Yaskawa INFORM job: R1_W27-A4(90,180)_KM_OKR2.JBI

/JOB
//NAME R1_W27-A4(90,180)_KM_OKR2
///FOLDERNAME KRIS-SCIANA
//POS
///NPOS 118,118,0,4,0,0
///TOOL 0
///POSTYPE PULSE
///PULSE
C00000=32571,-80067,-84751,-11816,58952,90735
C00001=-67595,-7768,-7207,-35750,73978,14125
C00002=-80598,-12710,-1030,-12842,70034,20340
C00003=-80599,-11861,1339,-12921,69037,20449
C00004=-81000,-11036,2695,-12887,68573,20352
C00005=-81299,-9950,3539,-12832,68562,20243
C00006=-81000,-11036,2695,-12887,68573,20352
C00007=-81000,-10543,4006,-12934,68033,20413
C00008=-81000,-11036,2695,-12887,68573,20352
C00009=-75972,290,11097,-17522,77040,34163
C00010=-77593,1159,14199,-17529,75300,33832
C00011=-78143,394,13556,-17496,75184,33650
C00012=-76339,27,10557,-17490,77151,34011
C00013=-80626,-11766,1412,-1925,55938,-1242
C00014=-80604,-16885,-14856,-12449,76250,19682
C00015=-77456,-22313,-19864,-6461,54131,78276
C00016=-80617,-11800,1386,-5311,46263,77368
C00017=-80614,-11811,1378,-5312,46263,77369
C00018=-78140,-17185,-212,-9910,41317,79160
C00019=-81168,-11680,2550,-5032,45575,77151
C00020=-80549,-12659,-567,-5287,47025,77356
C00021=-80487,-9351,5308,-7996,42180,77220
C00022=-80443,-11156,2742,-7947,42700,77191
C00023=-78226,-17049,-5584,-9114,45005,78042
C00024=-65420,23358,31165,-31257,71438,79494
C00025=-69378,27768,34519,-28549,68162,78619
C00026=-72413,51384,60505,-31158,65726,78265
C00027=-70611,42888,44989,-30390,70865,77539
C00028=-75134,-18461,-8114,-8268,49134,79639
C00029=-60313,-3477,16980,-41555,55752,85580
C00030=-62489,3761,29741,-43135,51633,86477
C00031=-62237,-78,28693,-47808,49629,88321
C00032=-72725,-17442,16408,-48318,42887,86419
C00033=-73223,-18395,15173,-47971,42820,86127
C00034=-67567,-15084,22766,-58607,48988,88210
C00035=-63268,-16746,16437,-56715,53119,87678
C00036=-77858,-27328,-27234,-6102,56048,77996
C00037=-77858,-27328,-27234,-6102,56048,-8278
C00038=-80560,-12001,1232,-23099,89880,39412
C00039=-80562,-11997,1235,-23099,89879,39412
C00040=-78546,-18752,-3942,-25358,87679,36764
C00041=-80047,-13896,-475,-23041,90092,39558
C00042=-79798,-10562,2405,-23011,90108,39646
C00043=-73705,-22874,2066,-31104,79210,44816
C00044=-72021,-22899,-1394,-31558,81149,45389
C00045=-88031,-25229,-22330,-24784,80292,46149
C00046=-74088,-81304,-57132,-46161,69139,49662
C00047=-13751,-81304,-57132,-46161,69139,49662
C00048=-24109,-97173,-75461,34297,58935,85832
C00049=-132100,-97173,-75461,34297,58935,85832
C00050=-132100,-17749,-28309,34297,58935,85832
C00051=-141655,18569,18708,54034,61749,83780
C00052=-140768,20217,21001,54093,60893,83749
C00053=-140768,20800,22898,54481,60371,83384
C00054=-140768,20217,21001,54093,60893,83749
C00055=-155664,19548,-11523,52673,81534,88020
C00056=-155140,18902,-12130,52523,81276,88141
C00057=-155664,19548,-11523,52673,81534,88020
C00058=-158287,-5700,5569,105477,62147,36289
C00059=-144891,17092,-14804,43908,85975,-9420
C00060=-144769,18045,-13920,43877,85878,-9408
C00061=-144891,17092,-14804,43908,85975,-9420
C00062=-120685,-15702,-31365,37390,69929,-5219
C00063=-125243,-75050,-65186,41337,64400,-9516
C00064=-90896,-91458,-74251,-13136,53772,27340
C00065=-85987,-45741,-53209,-41665,69322,45489
C00066=-80494,-11458,-25164,-47215,58644,80185
C00067=-84628,7522,-7873,-39732,61287,77186
C00068=-84628,7527,-7756,-39756,61234,77209
C00069=-84628,7615,-6294,-40053,60572,77489
C00070=-84628,7527,-7756,-39756,61234,77209
C00071=-85256,7794,-7522,-39492,60943,77025
C00072=-84628,7527,-7756,-39756,61234,77209
C00073=-84548,-2953,-19505,-38708,62473,76294
C00074=-89907,-10175,-21479,-33907,55460,73341
C00075=-87623,10863,-3696,-31122,53378,71592
C00076=-84515,20655,5407,-36942,57155,75370
C00077=-78402,3649,-16519,-40799,66441,77543
C00078=-80660,6683,-13306,-40007,65091,-11870
C00079=-73617,-18498,-32420,-43032,67485,-9563
C00080=-69872,-48029,-51657,-45224,66900,-7445
C00081=-99316,-51390,-56534,-3784,56840,-8136
C00082=-108651,-54845,-55282,14011,52033,-11284
C00083=-128597,-2477,-24064,39626,75198,-6696
C00084=-106236,880,-10934,32720,60711,-2021
C00085=-100502,752,-10642,30155,58374,-188
C00086=-121335,-12341,949,71341,33536,66986
C00087=-121314,-12325,1002,51085,42465,78387
C00088=-121322,-12342,996,51093,42465,78381
C00089=-120884,-12665,812,50951,42190,78492
C00090=-121319,-13000,-806,50447,42963,78778
C00091=-122361,-12330,1002,51521,43046,78059
C00092=-121327,-12349,995,51098,42466,78378
C00093=-121327,-12349,995,51098,42466,78378
C00094=-121328,-12349,996,51099,42466,78378
C00095=-121325,-12342,998,51095,42466,78380
C00096=-121317,-12324,1004,51087,42465,78386
C00097=-121324,-12328,964,64351,35558,70777
C00098=-121305,-12313,996,32749,35201,-57468
C00099=-121211,-12064,797,41015,45464,-52570
C00100=-117301,-7988,606,30593,47867,-49050
C00101=-116538,-6009,3661,32359,46841,-49122
C00102=-121892,-12966,-560,41565,45795,-52476
C00103=-122357,-12481,889,42191,45531,-52907
C00104=-118375,1792,12378,38125,46112,-50726
C00105=-117383,2243,11183,34310,46791,-49685
C00106=-119475,-3356,5120,33593,48382,-50093
C00107=-123076,-14640,-755,42570,45804,-53197
C00108=-121299,-12321,1006,38012,34307,-57526
C00109=-116680,1248,11585,32129,38176,11345
C00110=-123012,14798,28982,55920,47572,8352
C00111=-118370,22214,39637,57006,43279,8118
C00112=-115461,22065,39512,56211,41576,8915
C00113=-120097,15317,31288,56093,45198,8516
C00114=-131063,-13667,3794,57031,52830,6808
C00115=-129161,-95207,-43414,62198,28328,-70913
C00116=-59909,-164103,-90939,63385,27988,-71515
C00117=-83,-164103,-90939,8908,68191,-71515
BC00000=130065,689852,1043460
BC00001=112824,718177,1070908
BC00002=111165,751794,1070910
BC00003=110061,756556,1060794
BC00004=109620,758461,1052490
BC00005=109620,758461,1052490
BC00006=109620,758461,1052490
BC00007=109620,758461,1052490
BC00008=109620,758461,1052490
BC00009=120151,759047,1049688
BC00010=120151,759047,1049688
BC00011=120151,759047,1049688
BC00012=120151,759047,1049688
BC00013=70060,741920,1053417
BC00014=111165,751794,1070910
BC00015=83169,742337,1070910
BC00016=82698,742428,1048015
BC00017=82641,744606,1022235
BC00018=82618,745477,1011923
BC00019=82618,745477,1011923
BC00020=82618,745477,1011923
BC00021=82618,745477,1011923
BC00022=82618,745477,1011923
BC00023=82618,745477,1011923
BC00024=82618,745477,1011923
BC00025=82618,745477,1011923
BC00026=82618,745477,1011923
BC00027=82618,745477,1011923
BC00028=83161,750209,1070909
BC00029=83161,750209,1070909
BC00030=83161,750209,1070909
BC00031=83161,750209,1070909
BC00032=83161,750209,1070909
BC00033=83161,750209,1070909
BC00034=83161,750209,1070909
BC00035=83161,750209,1070909
BC00036=83169,742337,1070910
BC00037=83169,742337,1070910
BC00038=163703,784171,1043682
BC00039=158492,786234,1024678
BC00040=156487,787029,1017362
BC00041=156407,787060,1017077
BC00042=156407,787060,1017077
BC00043=156415,787057,1017105
BC00044=156407,787060,1017077
BC00045=170469,758461,974941
BC00046=163703,784171,1043682
BC00047=61771,679181,1043682
BC00048=85545,676876,144252
BC00049=233984,676876,144252
BC00050=233984,680564,144252
BC00051=262714,720037,211879
BC00052=262714,720037,211879
BC00053=262714,720037,211879
BC00054=262714,720037,211879
BC00055=308586,730328,18317
BC00056=308586,730328,18317
BC00057=308586,730328,18317
BC00058=299911,725264,31418
BC00059=290428,719729,45738
BC00060=290428,719729,45738
BC00061=290428,719729,45738
BC00062=200947,733780,116006
BC00063=194071,727260,112331
BC00064=194071,733780,131686
BC00065=194071,733780,131686
BC00066=142355,733775,131685
BC00067=142355,733775,131685
BC00068=142355,733775,131685
BC00069=142355,733775,131685
BC00070=142355,733775,131685
BC00071=142355,733775,131685
BC00072=142355,733775,131685
BC00073=142839,733745,131500
BC00074=142839,733745,131500
BC00075=142839,733745,131500
BC00076=142839,733745,131500
BC00077=142839,733745,131500
BC00078=142839,733745,131500
BC00079=142839,733745,131500
BC00080=142839,733745,131500
BC00081=185847,731066,115033
BC00082=185847,731066,115033
BC00083=232987,728130,96983
BC00084=175420,736488,148318
BC00085=159305,737658,155504
BC00086=192613,686942,193845
BC00087=213838,737567,276194
BC00088=219104,740206,258265
BC00089=221210,741261,251094
BC00090=221210,741261,251094
BC00091=221210,741261,251094
BC00092=221201,745870,251100
BC00093=221200,746303,251100
BC00094=221190,750911,251106
BC00095=219084,749856,258278
BC00096=213818,747217,276207
BC00097=195218,691822,223843
BC00098=207171,709248,282440
BC00099=215795,751561,279449
BC00100=215795,751561,279449
BC00101=215795,751561,279449
BC00102=222566,755703,266568
BC00103=222566,755703,266568
BC00104=215795,751561,279449
BC00105=215795,751561,279449
BC00106=215795,751561,279449
BC00107=213454,758065,282759
BC00108=216823,707918,296192
BC00109=216823,707918,296192
BC00110=216823,707918,296192
BC00111=216823,707918,296192
BC00112=216823,707918,296192
BC00113=216823,707918,296192
BC00114=216823,707918,296192
BC00115=216823,707918,296192
BC00116=216823,707918,296192
BC00117=119332,707918,853819
///POSTYPE BASE
///RECTAN
///RCONF 0,0,0,0,0,0,0,0,0,0,0,0,0,0,0,0,0,0,0,0,0,0,0,0
P00006=0.222,-3.123,-1.508,0.0000,0.0000,0.0000
P00014=-0.708,0.505,-8.393,0.0000,0.0000,0.0000
P00021=-0.225,-6.128,-0.405,0.0000,0.0000,0.0000
P00030=5.926,-4.294,-1.390,0.0000,0.0000,0.0000
//INST
///DATE 2024/07/25 10:56
///ATTR SC,RW
///GROUP1 RB1,BS1
NOP
'r2_W27-A4(90,180)
'
'Path S896
SFTOF
MOVJ C00000 BC00000 VJ=50.00
MOVJ C00001 BC00001 VJ=50.00
MOVL C00002 BC00002 V=100.0
MOVL C00003 BC00003 V=100.0
MOVL C00004 BC00004 V=60.0
REFP 3 C00005 BC00005
CALL JOB:SEARCH-R1
SET P014 P006
SFTON P014
MOVL C00006 BC00006 V=100.0
REFP 3 C00007 BC00007
CALL JOB:SEARCH-R1
SET P014 P006
SFTON P014
MOVL C00008 BC00008 V=100.0
MOVL C00009 BC00009 V=100.0
MOVL C00010 BC00010 V=100.0
REFP 3 C00011 BC00011
CALL JOB:SEARCH-R1
SET P014 P006
SFTON P014
MOVL C00012 BC00012 V=100.0
MOVL C00013 BC00013 V=100.0
'Path VIA902
SFTOF
MOVJ C00014 BC00014 VJ=20.00
'Path W898
SFTOF
SFTON P014
MOVJ C00015 BC00015 VJ=20.00
MOVJ C00016 BC00016 VJ=20.00
MOVL C00017 BC00017 V=100.0
MOVL C00018 BC00018 V=166.7 PL=0
REFP 1 C00019 BC00019
REFP 2 C00020 BC00020
MACRO1 MJ#(0) ARGF7
ARCON
MOVL C00021 BC00021 V=10.0
ARCOF
MOVL C00022 BC00022 V=166.7
MOVL C00023 BC00023 V=166.7
SFTON P014
MOVL C00024 BC00024 V=83.3
ARCON
MOVL C00025 BC00025 V=9.2
ARCON
MOVL C00026 BC00026 V=9.2
ARCOF
MOVL C00027 BC00027 V=200.0
MOVL C00028 BC00028 V=400.0
SFTOF
MOVJ C00029 BC00029 VJ=20.00
SFTON P014
MOVJ C00030 BC00030 VJ=10.00
ARCON
MOVL C00031 BC00031 V=9.2
MOVL C00032 BC00032 V=9.2
MOVL C00033 BC00033 V=9.2
MOVL C00034 BC00034 V=9.2
ARCOF
MOVJ C00035 BC00035 VJ=10.00
'Path VIA903
SFTOF
MOVJ C00036 BC00036 VJ=20.00
'Path VIA904
SFTOF
MOVJ C00037 BC00037 VJ=20.00
'Path W901
SFTOF
SFTON P014
MOVJ C00038 BC00038 VJ=20.00
MOVL C00039 BC00039 V=100.0
MOVL C00040 BC00040 V=100.0 PL=0
REFP 1 C00041 BC00041
REFP 2 C00042 BC00042
MACRO1 MJ#(0) ARGF6
ARCON
MOVL C00043 BC00043 V=11.7
ARCOF
MOVL C00044 BC00044 V=100.0
MOVL C00045 BC00045 V=100.0
SFTOF
'Path VIA907
SFTOF
MOVJ C00046 BC00046 VJ=20.00
'Path VIA905
SFTOF
MOVJ C00047 BC00047 VJ=100.00
CALL JOB:CLEAN-R1_KM_NEW_SCIANA
'Path VIA906
SFTOF
MOVJ C00048 BC00048 VJ=50.00
MOVJ C00049 BC00049 VJ=100.00
'Path S845
SFTOF
MOVJ C00050 BC00050 VJ=50.00
MOVL C00051 BC00051 V=133.3
MOVL C00052 BC00052 V=60.0
REFP 3 C00053 BC00053
CALL JOB:SEARCH-R1
SET P021 P006
SFTON P021
MOVL C00054 BC00054 V=60.0
MOVL C00055 BC00055 V=166.7
REFP 3 C00056 BC00056
CALL JOB:SEARCH-R1
SET P021 P006
SFTON P021
MOVL C00057 BC00057 V=100.0
MOVL C00058 BC00058 V=166.7
MOVL C00059 BC00059 V=100.0
REFP 3 C00060 BC00060
CALL JOB:SEARCH-R1
SET P021 P006
SFTON P021
MOVL C00061 BC00061 V=60.0
SFTOF
MOVJ C00062 BC00062 VJ=10.00
MOVJ C00063 BC00063 VJ=30.00
MOVJ C00064 BC00064 VJ=30.00
MOVJ C00065 BC00065 VJ=10.00
MOVJ C00066 BC00066 VJ=10.00
MOVJ C00067 BC00067 VJ=10.00
'POMIAR
MOVL C00068 BC00068 V=83.3
REFP 3 C00069 BC00069
CALL JOB:SEARCH-R1
SET P030 P006
SFTON P030
MOVL C00070 BC00070 V=83.3
REFP 3 C00071 BC00071
CALL JOB:SEARCH-R1
SET P030 P006
SFTON P030
MOVL C00072 BC00072 V=83.3
SFTOF
SFTON P030
MOVJ C00073 BC00073 VJ=10.00
MACRO1 MJ#(0) ARGF7
MOVJ C00074 BC00074 VJ=10.00
ARCON
MOVL C00075 BC00075 V=7.5
MOVL C00076 BC00076 V=7.5
ARCOF
MOVJ C00077 BC00077 VJ=15.00
SFTOF
MOVJ C00078 BC00078 VJ=20.00
MOVJ C00079 BC00079 VJ=20.00
MOVJ C00080 BC00080 VJ=20.00
MOVJ C00081 BC00081 VJ=30.00
MOVJ C00082 BC00082 VJ=30.00
MOVL C00083 BC00083 V=100.0
MOVL C00084 BC00084 V=100.0
MOVL C00085 BC00085 V=100.0
'Path W846
SFTOF
SFTON P021
MOVJ C00086 BC00086 VJ=20.00
MOVL C00087 BC00087 V=100.0
MOVL C00088 BC00088 V=166.7
MOVL C00089 BC00089 V=166.7 PL=0
REFP 1 C00090 BC00090
REFP 2 C00091 BC00091
MACRO1 MJ#(0) ARGF0
COMM ARCON
MOVL C00092 BC00092 V=10.0
MOVL C00093 BC00093 V=10.0
MOVL C00094 BC00094 V=10.0
ARCOF
MOVL C00095 BC00095 V=166.7
MOVL C00096 BC00096 V=250.0
MOVL C00097 BC00097 V=416.7
SFTOF
'Path W847
SFTOF
SFTON P021
MOVJ C00098 BC00098 VJ=20.00
MOVL C00099 BC00099 V=333.3
MOVL C00100 BC00100 V=166.7
MOVL C00101 BC00101 V=166.7 PL=0
REFP 1 C00102 BC00102
REFP 2 C00103 BC00103
MACRO1 MJ#(0) ARGF7
ARCON
MOVL C00104 BC00104 V=8.3
MOVL C00105 BC00105 V=8.3
ARCOF
SFTOF
MOVL C00106 BC00106 V=166.7
MOVL C00107 BC00107 V=250.0
MOVJ C00108 BC00108 VJ=20.00
MOVJ C00109 BC00109 VJ=30.00
MOVJ C00110 BC00110 VJ=20.00
MACRO1 MJ#(0) ARGF7
MOVJ C00111 BC00111 VJ=10.00
ARCON
MOVL C00112 BC00112 V=8.3
ARCOF
MOVJ C00113 BC00113 VJ=10.00
SFTOF
MOVJ C00114 BC00114 VJ=40.00
MOVJ C00115 BC00115 VJ=40.00
MOVJ C00116 BC00116 VJ=100.00
MOVJ C00117 BC00117 VJ=100.00
END
